PROGRAM MAIN
VAR
	m : INT;
END_VAR

m := m + 1;
PrgMqttCom();

END_PROGRAM

(* stored: Version 1.1.0.1, ProductVersion 3.1.4022.16
   POU MAIN: Id {f8d32ae9-13cf-4728-a76d-5f7c7fa15593}, SpecialFunc None *)
